// TIA Portal project "SCL PESCADERIA" (V11)

(* hardware
DEVICE "S7300/ET200 station_1"  SIMATIC 300-Station
   slot 0: "Perfil soporte_0"  Rail  6ES7 390-1***0-0AA0
   slot 2: "PLC_1"  CPU 313C-2 DP  6ES7 313-6CF03-0AB0  V2.6
      slot 0: "Interfaz MPI_1"  MPI
      slot 1: "Interfaz DP_1"  DP
      slot 2: "DI16/DO16_1"  DI16/DO16
      slot 4: "Contaje_1"  Counter
*)

// ===== PLC "PLC_1"  CPU 313C-2 DP =====

VAR_GLOBAL   // PLC tag table "Tabla de variables estándar"
   "Tag_1" AT %A0.0 : Bool;
   "Tag_2" AT %A0.1 : Bool;
   "Tag_3" AT %A0.2 : Bool;
   "Tag_4" AT %A0.3 : Bool;
   "Tag_5" AT %A0.4 : Bool;
   "Tag_6" AT %A0.5 : Bool;
   "Tag_7" AT %MD0 : Real;
   "Tag_8" AT %MD4 : Real;
   "Tag_9" AT %E0.0 : Bool;
   "Tag_10" AT %E0.1 : Bool;
   "Tag_11" AT %E0.2 : Bool;
   "Tag_12" AT %E0.3 : Bool;
   "Tag_13" AT %E0.4 : Bool;
   "Tag_14" AT %E0.5 : Bool;
END_VAR

DATA_BLOCK "PRECIOS_DB"   // DB1
{ S7_Optimized_Access := 'FALSE' }
VERSION : 0.1
// stored: InstanceOfName PRECIOS
"PRECIOS"
BEGIN
END_DATA_BLOCK

FUNCTION_BLOCK "PRECIOS"   // FB1, SCL
{ S7_Optimized_Access := 'FALSE' }
VERSION : 0.1
   VAR_INPUT
      ON : Bool;
      RESET : Bool;
      PESO : Real;
      SALMON : Bool;
      BOQUERONES : Bool;
      MELILLONES : Bool;
      BACALADILLA : Bool;
      IVA : Real;
   END_VAR
   VAR_OUTPUT
      "P BRUTO" : Real;
      "P NETO" : Real;
   END_VAR
   VAR
      "PVP SALMON" : Real;
      "PVP BOQUERONES" : Real;
      "PVP MEJILLONES" : Real;
      "PVP BACALADILLA" : Real;
      "PRECIO SALMON" : Real := 1.5;
      "PRECIO BOQUERONES" : Real := 3.8;
      "PRECIO MEJILLONES" : Real := 5.4;
      "PRECIO BACALADILLA" : Real := 3.4;
      "PT SALMON" : Real;
      "PT BOQUERONES" : Real;
      "PT MEJILLONES" : Real;
      "PT BACALADILLA" : Real;
      "IVA SALMON" : Real;
      "IVA BOQUERONES" : Real;
      "IVA MEJILLONES" : Real;
      "IVA BACALADILLA" : Real;
   END_VAR
BEGIN
   IF #RESET THEN (* puesta 0 marcadores y bloqueo de pulsadores *)
     #"P BRUTO":=0.0;
     #"P NETO" :=0.0;
     RETURN;
     END_IF;

     IF #ON AND #SALMON THEN (* pulsador salmon - marcador precio neto y bruto *)
       #"PVP SALMON" := #PESO * #"PRECIO SALMON" ;
       #"IVA SALMON":= #"PVP SALMON" * #IVA / 100.0 ;
        #"P NETO" := #PESO * #"PRECIO SALMON";    
       #"P BRUTO" := #"PVP SALMON" + #"IVA SALMON";
        END_IF;

   IF #ON AND #BOQUERONES THEN (* pulsador boquerones - marcador precio neto y bruto *)
       #"PVP BOQUERONES" := #PESO * #"PRECIO BOQUERONES" ;
       #"IVA BOQUERONES" := #"PVP BOQUERONES" * #IVA / 100.0 ;
        #"P NETO" := #PESO * #"PRECIO BOQUERONES";    
       #"P BRUTO" := #"PVP BOQUERONES" + #"IVA BOQUERONES";
     END_IF;

     IF #ON AND #MELILLONES THEN (* pulsador mejillones - marcador precio neto y bruto *)
       #"PVP MEJILLONES" := #PESO * #"PRECIO MEJILLONES" ;
       #"IVA MEJILLONES" := #"PVP MEJILLONES" * #IVA / 100.0 ;
        #"P NETO" := #PESO * #"PRECIO MEJILLONES"  ;    
       #"P BRUTO" := #"PVP MEJILLONES" + #"IVA MEJILLONES";
     END_IF;

     IF #ON AND #BACALADILLA THEN (* pulsador bacaladilla - marcador precio neto y bruto *)
       #"PVP BACALADILLA" := #PESO * #"PRECIO BACALADILLA" ;
       #"IVA BACALADILLA"  := #"PVP BACALADILLA" * #IVA / 100.0 ;
        #"P NETO" := #PESO * #"PRECIO BACALADILLA";    
        #"P BRUTO" := #"PVP BACALADILLA" + #"IVA BACALADILLA";
        END_IF;
END_FUNCTION_BLOCK

ORGANIZATION_BLOCK "Main"   // OB1, LAD
TITLE = "Main Program Sweep (Cycle)"
{ S7_Optimized_Access := 'FALSE' }
VERSION : 0.1
   VAR_TEMP
      OB1_EV_CLASS : Byte;   // Bits 0-3 = 1 (Coming event), Bits 4-7 = 1 (Event class 1)
      OB1_SCAN_1 : Byte;   // 1 (Cold restart scan 1 of OB 1), 3 (Scan 2-n of OB 1)
      OB1_PRIORITY : Byte;   // Priority of OB Execution
      OB1_OB_NUMBR : Byte;   // 1 (Organization block 1, OB1)
      OB1_RESERVED_1 : Byte;   // Reserved for system
      OB1_RESERVED_2 : Byte;   // Reserved for system
      OB1_PREV_CYCLE : Int;   // Cycle time of previous OB1 scan (milliseconds)
      OB1_MIN_CYCLE : Int;   // Minimum cycle time of OB1 (milliseconds)
      OB1_MAX_CYCLE : Int;   // Maximum cycle time of OB1 (milliseconds)
      OB1_DATE_TIME : Date_And_Time;   // Date and time OB1 started
   END_VAR
BEGIN

REGION Network 1
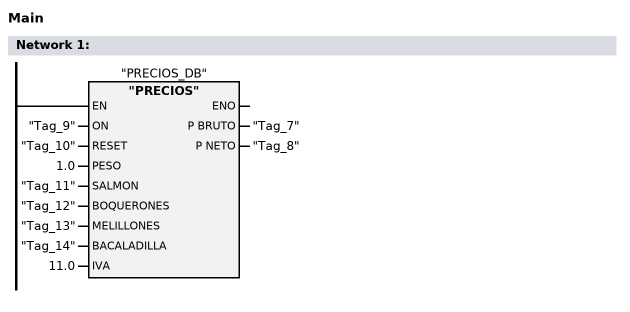
   RUNG wire#powerrail
      "PRECIOS_DB"(ON := "Tag_9", RESET := "Tag_10", PESO := 1.0, SALMON := "Tag_11", BOQUERONES := "Tag_12", MELILLONES := "Tag_13", BACALADILLA := "Tag_14", IVA := 11.0, "P BRUTO" => "Tag_7", "P NETO" => "Tag_8")
   END_RUNG
   // the same network as SCL:
   "PRECIOS_DB"(ON := "Tag_9",   // "PRECIOS"
                RESET := "Tag_10",
                PESO := 1.0,
                SALMON := "Tag_11",
                BOQUERONES := "Tag_12",
                MELILLONES := "Tag_13",
                BACALADILLA := "Tag_14",
                IVA := 11.0,
                "P BRUTO" => "Tag_7",
                "P NETO" => "Tag_8");
END_REGION
END_ORGANIZATION_BLOCK